FUNCTION_BLOCK StrapMachine
VAR_INPUT
	bEnable : BOOL;
END_VAR
VAR_OUTPUT
	enable AT %Q* : BOOL;
	execute AT %Q* : BOOL;
	reset AT %Q* : BOOL;
	
	error AT %I* : BOOL;
	ready AT %I* : BOOL;
	//busy (*AT %I**) : BOOL;
	done AT %I* : BOOL;
	home AT %I* : BOOL;
	
	timeout : BOOL;
	
	atBundleLevel AT %I* : BOOL;
END_VAR
VAR	
	holdPost : TON;
	delay : TON;
	
	start : BOOL;
	step : (SETUP, RUN, WAIT);
END_VAR
VAR_STAT CONSTANT
	pulseTime : TIME := T#100MS;
	holdTime : TIME := T#500MS;
	maxDelay : TIME := T#30S;
END_VAR

holdPost(IN:= , PT:= holdTime, Q=> , ET=> );
delay(IN:= step > 0 OR start, PT:= maxDelay, Q=> timeout, ET=> );

IF delay.Q THEN
	delay.IN := FALSE;
	//timeout := TRUE;
	//busy := FALSE;
	
	start := FALSE;
	step := SETUP;
END_IF

enable := bEnable AND robot1.strapSafetyIn AND robot2.strapSafetyIn;

CASE step OF
	SETUP:
		//busy := FALSE;
		IF error THEN
			enable := FALSE;
			execute := FALSE;
			clear();
			
		ELSIF start AND enable THEN //strapping does not start if error
			start := FALSE;
			step := RUN;
		END_IF
	
	RUN:
		IF NOT execute THEN
			execute := TRUE;
			RETURN; //keeps execute TRUE for at least 1 cycle
		END_IF
		
		IF execute AND NOT ready (*AND NOT home*) THEN
			execute := FALSE;
			step := WAIT;
		END_IF
		
	WAIT: //due to the use of DC motors instead of stepper motors in the machine, a short delay is required before next strap
		IF home THEN
			holdPost.IN := TRUE;
			enable := FALSE;
			execute := FALSE;
		END_IF
		
		IF holdPost.Q THEN
			holdPost.IN := FALSE;
			done := TRUE;
			step := 0;
		END_IF
		
END_CASE

(*
executePulse(IN:= , PT:= pulseTime, Q=> , ET=> );
execute := executePulse.IN AND NOT executePulse.Q;

IF executePulse.Q THEN
	executePulse.IN := FALSE;
END_IF


resetPulse(IN:= , PT:= pulseTime, Q=> , ET=> );
StrapMachineST.reset := resetPulse.IN AND NOT resetPulse.Q;

IF resetPulse.Q THEN
	executePulse.IN := FALSE;
END_IF

ready := enable AND NOT execute AND NOT StrapMachineST.reset AND NOT error AND home;
*)

METHOD clear : BOOL
VAR_INPUT
END_VAR
(*
reset should be continuously called until machine returns evidence that it is ready again
machine is expected to not respond to reset signals if it is already in an idle state
*)
enable := FALSE;
execute := FALSE;

IF error THEN
	reset := NOT reset;
ELSE
	reset := FALSE;
END_IF

clear := NOT error;
END_METHOD

METHOD strap : BOOL
VAR_INPUT
END_VAR
//IF ready AND NOT busy AND NOT error THEN
	//busy := TRUE;
	//start := TRUE;
	//strap := TRUE;
//END_IF

start := TRUE;
END_METHOD

END_FUNCTION_BLOCK

(* stored: Version 1.1.0.1, ProductVersion 3.1.4024.11
   POU StrapMachine: Id {195d23e9-3ade-4278-a206-bfe5b204b6b8}, SpecialFunc None
   Method clear: Id {6ec69dfe-8ae5-445c-9814-e61a9b3ae255}
   Method strap: Id {8221f6b6-4ed9-46c5-a2f2-3e9b4c2e4608} *)
